LIN {X 0,Y 99.538,Z 705.154,A -85,B 0,C 180,E1 -30433.877,E2 -30433.877} C_VEL
LIN {X 0,Y 92.855,Z 716.866,A -85,B 0,C 180,E1 -30435.204,E2 -30435.204} C_VEL
LIN {X 0,Y 85.443,Z 727.347,A -85,B 0,C 180,E1 -30437.026,E2 -30437.026} C_VEL
LIN {X 0,Y 78.023,Z 735.936,A -85,B 0,C 180,E1 -30438.956,E2 -30438.956} C_VEL
LIN {X 0,Y 73.258,Z 740.751,A -85,B 0,C 180,E1 -30440.398,E2 -30440.398} C_VEL
LIN {X 0,Y 68.907,Z 744.631,A -85,B 0,C 180,E1 -30441.253,E2 -30441.253} C_VEL
LIN {X 0,Y 60.889,Z 750.458,A -85,B 0,C 180,E1 -30441.745,E2 -30441.745} C_VEL
LIN {X 0,Y 52.484,Z 755.617,A -85,B 0,C 180,E1 -30442.685,E2 -30442.685} C_VEL
LIN {X 0,Y 47.586,Z 758.441,A -85,B 0,C 180,E1 -30444.648,E2 -30444.648} C_VEL
LIN {X 0,Y 37.586,Z 763.703,A -85,B 0,C 180,E1 -30452.71,E2 -30452.71} C_VEL
LIN {X 0,Y 29.331,Z 767.316,A -85,B 0,C 180,E1 -30464.044,E2 -30464.044} C_VEL
LIN {X 0,Y 24.819,Z 769.182,A -85,B 0,C 180,E1 -30475.506,E2 -30475.506} C_VEL
LIN {X 0,Y 21.517,Z 770.594,A -85,B 0,C 180,E1 -30490.936,E2 -30490.936} C_VEL
LIN {X 0,Y 20.011,Z 771.603,A -85,B 0,C 180,E1 -30510,E2 -30510} C_VEL
LIN {X 0,Y 20.655,Z 772.235,A -85,B 0,C 180,E1 -30529.892,E2 -30529.892} C_VEL
LIN {X 0,Y 23.357,Z 772.487,A -85,B 0,C 180,E1 -30546.998,E2 -30546.998} C_VEL
LIN {X 0,Y 27.522,Z 772.315,A -85,B 0,C 180,E1 -30560.002,E2 -30560.002} C_VEL
LIN {X 0,Y 38.503,Z 770.782,A -85,B 0,C 180,E1 -30575.871,E2 -30575.871} C_VEL
LIN {X 0,Y 48.032,Z 768.494,A -85,B 0,C 180,E1 -30582.983,E2 -30582.983} C_VEL
LIN {X 0,Y 57.585,Z 765.346,A -85,B 0,C 180,E1 -30587.511,E2 -30587.511} C_VEL
LIN {X 0,Y 67.62,Z 761.061,A -85,B 0,C 180,E1 -30590.876,E2 -30590.876} C_VEL
LIN {X 0,Y 77.842,Z 755.574,A -85,B 0,C 180,E1 -30593.271,E2 -30593.271} C_VEL
LIN {X 0,Y 88.618,Z 748.359,A -85,B 0,C 180,E1 -30595.451,E2 -30595.451} C_VEL
LIN {X 0,Y 98.534,Z 740.091,A -85,B 0,C 180,E1 -30596.899,E2 -30596.899} C_VEL
LIN {X 0,Y 107.245,Z 731.233,A -85,B 0,C 180,E1 -30597.918,E2 -30597.918} C_VEL
LIN {X 0,Y 115.11,Z 721.487,A -85,B 0,C 180,E1 -30598.709,E2 -30598.709} C_VEL
LIN {X 0,Y 122.116,Z 710.78,A -85,B 0,C 180,E1 -30599.354,E2 -30599.354} C_VEL
LIN {X 0,Y 128.126,Z 699.036,A -85,B 0,C 180,E1 -30599.946,E2 -30599.946} C_VEL
LIN {X 0,Y 130.018,Z 694.628,A -85,B 0,C 180,E1 -30600.085,E2 -30600.085} C_VEL
LIN {X 0,Y 130.609,Z 693.04,A -85,B 0,C 180,E1 -30600.77,E2 -30600.77} C_VEL
LIN {X 0,Y 130.649,Z 693.071,A -85,B 0,C 180,E1 -30603.083,E2 -30603.083} C_VEL
LIN {X 0,Y 130.252,Z 694.158,A -85,B 0,C 180,E1 -30603.435,E2 -30603.435} C_VEL
LIN {X 0,Y 125.016,Z 705.671,A -85,B 0,C 180,E1 -30603.78,E2 -30603.78} C_VEL
LIN {X 0,Y 118.91,Z 716.18,A -85,B 0,C 180,E1 -30604.174,E2 -30604.174} C_VEL
LIN {X 0,Y 111.078,Z 726.966,A -85,B 0,C 180,E1 -30604.799,E2 -30604.799} C_VEL
LIN {X 0,Y 102.39,Z 736.674,A -85,B 0,C 180,E1 -30605.586,E2 -30605.586} C_VEL
LIN {X 0,Y 93.733,Z 744.64,A -85,B 0,C 180,E1 -30606.564,E2 -30606.564} C_VEL
LIN {X 0,Y 83.394,Z 752.457,A -85,B 0,C 180,E1 -30608.028,E2 -30608.028} C_VEL
LIN {X 0,Y 71.449,Z 759.627,A -85,B 0,C 180,E1 -30610.387,E2 -30610.387} C_VEL
LIN {X 0,Y 61.586,Z 764.34,A -85,B 0,C 180,E1 -30613.192,E2 -30613.192} C_VEL
LIN {X 0,Y 51.502,Z 768.131,A -85,B 0,C 180,E1 -30617.215,E2 -30617.215} C_VEL
LIN {X 0,Y 45.077,Z 770.049,A -85,B 0,C 180,E1 -30620.701,E2 -30620.701} C_VEL
LIN {X 0,Y 38.896,Z 771.534,A -85,B 0,C 180,E1 -30625.389,E2 -30625.389} C_VEL
LIN {X 0,Y 27.84,Z 773.263,A -85,B 0,C 180,E1 -30640.771,E2 -30640.771} C_VEL
LIN {X 0,Y 23.556,Z 773.556,A -85,B 0,C 180,E1 -30653.367,E2 -30653.367} C_VEL
LIN {X 0,Y 20.759,Z 773.451,A -85,B 0,C 180,E1 -30670.212,E2 -30670.212} C_VEL
LIN {X 0,Y 20.017,Z 772.918,A -85,B 0,C 180,E1 -30690,E2 -30690} C_VEL
LIN {X 0,Y 20.749,Z 771.968,A -85,B 0,C 180,E1 -30709.799,E2 -30709.799} C_VEL
LIN {X 0,Y 23.496,Z 770.618,A -85,B 0,C 180,E1 -30726.743,E2 -30726.743} C_VEL
LIN {X 0,Y 30.244,Z 767.756,A -85,B 0,C 180,E1 -30744.42,E2 -30744.42} C_VEL
LIN {X 0,Y 38.788,Z 763.866,A -85,B 0,C 180,E1 -30754.948,E2 -30754.948} C_VEL
LIN {X 0,Y 48.155,Z 758.844,A -85,B 0,C 180,E1 -30761.555,E2 -30761.555} C_VEL
LIN {X 0,Y 57.904,Z 752.525,A -85,B 0,C 180,E1 -30766.158,E2 -30766.158} C_VEL
LIN {X 0,Y 67.906,Z 744.599,A -85,B 0,C 180,E1 -30769.48,E2 -30769.48} C_VEL
LIN {X 0,Y 76.395,Z 736.529,A -85,B 0,C 180,E1 -30771.464,E2 -30771.464} C_VEL
LIN {X 0,Y 84.96,Z 726.681,A -85,B 0,C 180,E1 -30773.043,E2 -30773.043} C_VEL
LIN {X 0,Y 92.721,Z 715.684,A -85,B 0,C 180,E1 -30774.162,E2 -30774.162} C_VEL
LIN {X 0,Y 99.543,Z 703.337,A -85,B 0,C 180,E1 -30774.977,E2 -30774.977} C_VEL
LIN {X 0,Y 104.869,Z 690.656,A -85,B 0,C 180,E1 -30775.599,E2 -30775.599} C_VEL
LIN {X 0,Y 108.646,Z 677.951,A -85,B 0,C 180,E1 -30775.996,E2 -30775.996} C_VEL
LIN {X 0,Y 110.002,Z 671.598,A -85,B 0,C 180,E1 -30776.223,E2 -30776.223} C_VEL
LIN {X 0,Y 109.889,Z 670.137,A -85,B 0,C 180,E1 -30778.626,E2 -30778.626} C_VEL
LIN {X 0,Y 109.842,Z 669.662,A -85,B 0,C 180,E1 -30780,E2 -30780} C_VEL
LIN {X 0,Y 109.785,Z 669.762,A -85,B 0,C 180,E1 -30784.13,E2 -30784.13} C_VEL
LIN {X 0,Y 109.918,Z 671.412,A -85,B 0,C 180,E1 -30787.847,E2 -30787.847} C_VEL
LIN {X 0,Y 109.947,Z 671.667,A -85,B 0,C 180,E1 -30788.257,E2 -30788.257} C_VEL
LIN {X 0,Y 107.13,Z 683.24,A -85,B 0,C 180,E1 -30788.643,E2 -30788.643} C_VEL
LIN {X 0,Y 102.756,Z 695.759,A -85,B 0,C 180,E1 -30789.271,E2 -30789.271} C_VEL
LIN {X 0,Y 97.22,Z 707.419,A -85,B 0,C 180,E1 -30789.963,E2 -30789.963} C_VEL
LIN {X 0,Y 90.414,Z 718.722,A -85,B 0,C 180,E1 -30791.086,E2 -30791.086} C_VEL
LIN {X 0,Y 82.804,Z 728.913,A -85,B 0,C 180,E1 -30792.567,E2 -30792.567} C_VEL
LIN {X 0,Y 74.336,Z 738.087,A -85,B 0,C 180,E1 -30794.293,E2 -30794.293} C_VEL
LIN {X 0,Y 65.954,Z 745.653,A -85,B 0,C 180,E1 -30796.462,E2 -30796.462} C_VEL
LIN {X 0,Y 56.16,Z 753.052,A -85,B 0,C 180,E1 -30800.191,E2 -30800.191} C_VEL
LIN {X 0,Y 47.586,Z 758.441,A -85,B 0,C 180,E1 -30804.648,E2 -30804.648} C_VEL
LIN {X 0,Y 42.61,Z 761.064,A -85,B 0,C 180,E1 -30807.039,E2 -30807.039} C_VEL
LIN {X 0,Y 33.585,Z 764.814,A -85,B 0,C 180,E1 -30809.853,E2 -30809.853} C_VEL
LIN {X 0,Y 26.224,Z 767.303,A -85,B 0,C 180,E1 -30813.33,E2 -30813.33} C_VEL
LIN {X 0,Y 21.112,Z 768.883,A -85,B 0,C 180,E1 -30819.493,E2 -30819.493} C_VEL
LIN {X 0,Y 19.633,Z 769.36,A -85,B 0,C 180,E1 -30822.877,E2 -30822.877} C_VEL
LIN {X 0,Y 14.987,Z 770.84,A -85,B 0,C 180,E1 -30842.035,E2 -30842.035} C_VEL
LIN {X 0,Y 12.913,Z 771.837,A -85,B 0,C 180,E1 -30870,E2 -30870} C_VEL
LIN {X 0,Y 14.169,Z 772.457,A -85,B 0,C 180,E1 -30899.735,E2 -30899.735} C_VEL
LIN {X 0,Y 18.156,Z 772.695,A -85,B 0,C 180,E1 -30920.73,E2 -30920.73} C_VEL
LIN {X 0,Y 29.698,Z 771.919,A -85,B 0,C 180,E1 -30941.185,E2 -30941.185} C_VEL
LIN {X 0,Y 42.828,Z 769.576,A -85,B 0,C 180,E1 -30949.919,E2 -30949.919} C_VEL
LIN {X 0,Y 53.034,Z 766.678,A -85,B 0,C 180,E1 -30953.648,E2 -30953.648} C_VEL
LIN {X 0,Y 63.385,Z 762.738,A -85,B 0,C 180,E1 -30956.265,E2 -30956.265} C_VEL
LIN {X 0,Y 75.583,Z 756.641,A -85,B 0,C 180,E1 -30958.293,E2 -30958.293} C_VEL
LIN {X 0,Y 86.089,Z 749.971,A -85,B 0,C 180,E1 -30959.81,E2 -30959.81} C_VEL
LIN {X 0,Y 96.645,Z 741.671,A -85,B 0,C 180,E1 -30960.901,E2 -30960.901} C_VEL
LIN {X 0,Y 98.406,Z 740.062,A -85,B 0,C 180,E1 -30961.048,E2 -30961.048} C_VEL
LIN {X 0,Y 98.438,Z 740.057,A -85,B 0,C 180,E1 -30961.803,E2 -30961.803} C_VEL
LIN {X 0,Y 87.942,Z 748.75,A -85,B 0,C 180,E1 -30962.649,E2 -30962.649} C_VEL
LIN {X 0,Y 77.471,Z 755.695,A -85,B 0,C 180,E1 -30963.737,E2 -30963.737} C_VEL
LIN {X 0,Y 67.044,Z 761.273,A -85,B 0,C 180,E1 -30965.233,E2 -30965.233} C_VEL
LIN {X 0,Y 56.701,Z 765.67,A -85,B 0,C 180,E1 -30967.444,E2 -30967.444} C_VEL
LIN {X 0,Y 49.863,Z 768.001,A -85,B 0,C 180,E1 -30969.389,E2 -30969.389} C_VEL
LIN {X 0,Y 43.076,Z 769.907,A -85,B 0,C 180,E1 -30971.789,E2 -30971.789} C_VEL
LIN {X 0,Y 36.413,Z 771.368,A -85,B 0,C 180,E1 -30975.201,E2 -30975.201} C_VEL
LIN {X 0,Y 29.915,Z 772.411,A -85,B 0,C 180,E1 -30980,E2 -30980} C_VEL
LIN {X 0,Y 18.341,Z 773.356,A -85,B 0,C 180,E1 -30999.972,E2 -30999.972} C_VEL
LIN {X 0,Y 14.264,Z 773.229,A -85,B 0,C 180,E1 -31020.483,E2 -31020.483} C_VEL
LIN {X 0,Y 12.924,Z 772.685,A -85,B 0,C 180,E1 -31050,E2 -31050} C_VEL
LIN {X 0,Y 14.251,Z 771.723,A -85,B 0,C 180,E1 -31079.548,E2 -31079.548} C_VEL
LIN {X 0,Y 18.293,Z 770.361,A -85,B 0,C 180,E1 -31100.206,E2 -31100.206} C_VEL
LIN {X 0,Y 26.728,Z 767.475,A -85,B 0,C 180,E1 -31116.966,E2 -31116.966} C_VEL
LIN {X 0,Y 36.35,Z 763.56,A -85,B 0,C 180,E1 -31125.172,E2 -31125.172} C_VEL
LIN {X 0,Y 46.395,Z 758.511,A -85,B 0,C 180,E1 -31129.932,E2 -31129.932} C_VEL
LIN {X 0,Y 53.634,Z 754.113,A -85,B 0,C 180,E1 -31132.471,E2 -31132.471} C_VEL
LIN {X 0,Y 63.509,Z 747.022,A -85,B 0,C 180,E1 -31134.824,E2 -31134.824} C_VEL
LIN {X 0,Y 73.925,Z 737.856,A -85,B 0,C 180,E1 -31136.564,E2 -31136.564} C_VEL
LIN {X 0,Y 83.519,Z 727.248,A -85,B 0,C 180,E1 -31137.757,E2 -31137.757} C_VEL
LIN {X 0,Y 91.393,Z 716.453,A -85,B 0,C 180,E1 -31138.495,E2 -31138.495} C_VEL
LIN {X 0,Y 97.527,Z 705.957,A -85,B 0,C 180,E1 -31138.961,E2 -31138.961} C_VEL
LIN {X 0,Y 103.01,Z 693.858,A -85,B 0,C 180,E1 -31139.366,E2 -31139.366} C_VEL
LIN {X 0,Y 107.323,Z 680.898,A -85,B 0,C 180,E1 -31139.682,E2 -31139.682} C_VEL
LIN {X 0,Y 108.358,Z 676.77,A -85,B 0,C 180,E1 -31139.859,E2 -31139.859} C_VEL
LIN {X 0,Y 108.286,Z 676.848,A -85,B 0,C 180,E1 -31144.226,E2 -31144.226} C_VEL
LIN {X 0,Y 108.277,Z 676.998,A -85,B 0,C 180,E1 -31144.642,E2 -31144.642} C_VEL
LIN {X 0,Y 104.625,Z 689.392,A -85,B 0,C 180,E1 -31145.07,E2 -31145.07} C_VEL
LIN {X 0,Y 99.41,Z 701.946,A -85,B 0,C 180,E1 -31145.532,E2 -31145.532} C_VEL
LIN {X 0,Y 93.651,Z 712.595,A -85,B 0,C 180,E1 -31146.112,E2 -31146.112} C_VEL
LIN {X 0,Y 85.872,Z 724.049,A -85,B 0,C 180,E1 -31147.106,E2 -31147.106} C_VEL
LIN {X 0,Y 78.098,Z 733.29,A -85,B 0,C 180,E1 -31148.168,E2 -31148.168} C_VEL
LIN {X 0,Y 69.464,Z 741.723,A -85,B 0,C 180,E1 -31149.451,E2 -31149.451} C_VEL
LIN {X 0,Y 59.21,Z 749.93,A -85,B 0,C 180,E1 -31151.703,E2 -31151.703} C_VEL
LIN {X 0,Y 50.755,Z 755.54,A -85,B 0,C 180,E1 -31154.244,E2 -31154.244} C_VEL
LIN {X 0,Y 40.764,Z 761.016,A -85,B 0,C 180,E1 -31158.52,E2 -31158.52} C_VEL
LIN {X 0,Y 31.088,Z 765.315,A -85,B 0,C 180,E1 -31165.277,E2 -31165.277} C_VEL
LIN {X 0,Y 24.935,Z 767.597,A -85,B 0,C 180,E1 -31172.271,E2 -31172.271} C_VEL
LIN {X 0,Y 19.633,Z 769.36,A -85,B 0,C 180,E1 -31182.877,E2 -31182.877} C_VEL
LIN {X 0,Y 16.781,Z 770.295,A -85,B 0,C 180,E1 -31190.924,E2 -31190.924} C_VEL
LIN {X 0,Y 12.531,Z 771.426,A -85,B 0,C 180,E1 -31206.691,E2 -31206.691} C_VEL
LIN {X 0,Y 8.775,Z 772.589,A -85,B 0,C 180,E1 -31258.63,E2 -31258.63} C_VEL
LIN {X 0,Y 12.723,Z 772.902,A -85,B 0,C 180,E1 -31297.145,E2 -31297.145} C_VEL
LIN {X 0,Y 16.166,Z 772.855,A -85,B 0,C 180,E1 -31305.233,E2 -31305.233} C_VEL
LIN {X 0,Y 28.215,Z 772.097,A -85,B 0,C 180,E1 -31315.082,E2 -31315.082} C_VEL
LIN {X 0,Y 35.167,Z 771.114,A -85,B 0,C 180,E1 -31317.724,E2 -31317.724} C_VEL
LIN {X 0,Y 44.082,Z 769.243,A -85,B 0,C 180,E1 -31319.999,E2 -31319.999} C_VEL
LIN {X 0,Y 49.2,Z 767.865,A -85,B 0,C 180,E1 -31320.851,E2 -31320.851} C_VEL
LIN {X 0,Y 49.205,Z 767.87,A -85,B 0,C 180,E1 -31321.175,E2 -31321.175} C_VEL
LIN {X 0,Y 42.2,Z 769.763,A -85,B 0,C 180,E1 -31322.268,E2 -31322.268} C_VEL
LIN {X 0,Y 35.223,Z 771.202,A -85,B 0,C 180,E1 -31323.944,E2 -31323.944} C_VEL
LIN {X 0,Y 21.442,Z 772.886,A -85,B 0,C 180,E1 -31330.488,E2 -31330.488} C_VEL
LIN {X 0,Y 14.811,Z 773.157,A -85,B 0,C 180,E1 -31338.378,E2 -31338.378} C_VEL
LIN {X 0,Y 8.805,Z 773.007,A -85,B 0,C 180,E1 -31357.041,E2 -31357.041} C_VEL
LIN {X 0,Y 5.818,Z 772.452,A -85,B 0,C 180,E1 -31410,E2 -31410} C_VEL
LIN {X 0,Y 8.793,Z 771.478,A -85,B 0,C 180,E1 -31463.056,E2 -31463.056} C_VEL
LIN {X 0,Y 14.782,Z 770.104,A -85,B 0,C 180,E1 -31481.966,E2 -31481.966} C_VEL
LIN {X 0,Y 24.822,Z 767.194,A -85,B 0,C 180,E1 -31492.291,E2 -31492.291} C_VEL
LIN {X 0,Y 35.207,Z 763.255,A -85,B 0,C 180,E1 -31496.45,E2 -31496.45} C_VEL
LIN {X 0,Y 47.443,Z 757.194,A -85,B 0,C 180,E1 -31499.135,E2 -31499.135} C_VEL
LIN {X 0,Y 57.983,Z 750.539,A -85,B 0,C 180,E1 -31500.64,E2 -31500.64} C_VEL
LIN {X 0,Y 68.553,Z 742.272,A -85,B 0,C 180,E1 -31501.733,E2 -31501.733} C_VEL
LIN {X 0,Y 77.368,Z 733.821,A -85,B 0,C 180,E1 -31502.295,E2 -31502.295} C_VEL
LIN {X 0,Y 77.411,Z 733.76,A -85,B 0,C 180,E1 -31502.987,E2 -31502.987} C_VEL
LIN {X 0,Y 66.908,Z 743.621,A -85,B 0,C 180,E1 -31503.752,E2 -31503.752} C_VEL
LIN {X 0,Y 56.451,Z 751.532,A -85,B 0,C 180,E1 -31505.15,E2 -31505.15} C_VEL
LIN {X 0,Y 46.022,Z 757.869,A -85,B 0,C 180,E1 -31506.976,E2 -31506.976} C_VEL
LIN {X 0,Y 35.652,Z 762.901,A -85,B 0,C 180,E1 -31509.73,E2 -31509.73} C_VEL
LIN {X 0,Y 25.382,Z 766.815,A -85,B 0,C 180,E1 -31514.282,E2 -31514.282} C_VEL
LIN {X 0,Y 15.396,Z 769.709,A -85,B 0,C 180,E1 -31524.084,E2 -31524.084} C_VEL
LIN {X 0,Y 9.341,Z 771.084,A -85,B 0,C 180,E1 -31541.204,E2 -31541.204} C_VEL
LIN {X 0,Y 5.804,Z 772.071,A -85,B 0,C 180,E1 -31590,E2 -31590} C_VEL
LIN {X 0,Y 8.719,Z 772.681,A -85,B 0,C 180,E1 -31643.713,E2 -31643.713} C_VEL
LIN {X 0,Y 16.166,Z 772.855,A -85,B 0,C 180,E1 -31665.233,E2 -31665.233} C_VEL
LIN {X 0,Y 16.166,Z 772.855,A -85,B 0,C 180,E1 -31665.233,E2 -31665.233}

QRS_NEXT_CUT()

QRS_NEXT()
QRS_HOME()

END
